INTERFACE INTERNAL I_ExecuteNode EXTENDS Debug.I_Debug;

METHOD INTERNAL Attach : Results.Result
VAR_INPUT
	iExecute		: I_ExecuteNode;
END_VAR
END_METHOD

METHOD INTERNAL Exe
VAR_INPUT
END_VAR
END_METHOD

PROPERTY INTERNAL state : Results.Result
GET
END_GET
SET
END_SET
END_PROPERTY

END_INTERFACE

(* stored: Version 1.1.0.1
   Itf I_ExecuteNode: Id {64b208cb-edd6-4de3-aa56-5a7326d6049a}
   Method Attach: Id {0ebe16bf-357a-4712-b807-2b68725d85b2}
   Method Exe: Id {08feb7a6-d2d3-4ecf-8c26-1ab33ca7e834}
   Property state: Id {d80d2393-ee18-4d5d-9b8c-78ec1518be37}
   Get Get: Id {db96e9af-bbbc-48f9-a856-70a64f30305d}
   Set Set: Id {0a7a2f5b-ce62-4bf5-b4e0-b6f6b9ee71b6} *)
